Yaskawa INFORM job: SET-SPINDLE.JBI

/JOB
//NAME SET-SPINDLE
//POS
///NPOS 0,0,0,0,0,0
//INST
///DATE 2025/10/24 13:58
///ATTR SC,RW
///GROUP1 RB1
NOP
'SET SPINDLE RPM
SET I003  EXPRESS I002 * 1.365 / 2340 * 100
AOUT AO#(1) I003
GETREG I000 MREG#(560) LOW
SET B000 I000
GETREG I001 MREG#(560) HIGH
SET B001 I001
DOUT OG#(20) B000
DOUT OG#(21) B001
END
